// TIA Portal V17 export
// export: Created 2023-02-13T11:16:20.9592979Z, ExportSetting WithDefaults, DisplayName Totally Integrated Automation Portal, DisplayVersion V17, DisplayName TIA Portal Openness, DisplayVersion V17, DisplayName TIA Portal Teamcenter Gateway, DisplayVersion V17, DisplayName TIA Portal Version Control Interface, DisplayVersion V17, DisplayName SINAMICS Startdrive Advanced, DisplayVersion V17, DisplayName SINAMICS Startdrive G130, G150, S120, S150, SINAMICS MV, S210, DisplayVersion V17, DisplayName SINAMICS Startdrive G110M, G120, G120C, G120D, G120P, G115D, DisplayVersion V17, DisplayName STEP 7 Professional, DisplayVersion V17, DisplayName STEP 7 Safety, DisplayVersion V17, DisplayName WinCC Professional, DisplayVersion V17
DATA_BLOCK "IO Digital Blending_DB"   // DB7
VERSION : 0.1
// stored: AutoNumber true, DBAccessibleFromOPCUA true, DBAccessibleFromWebserver true, InstanceOfName IO Digital Blending, InstanceOfType FB
"IO Digital Blending"
   // VAR_INPUT
   //    Init : Bool;
   //    Reset : Bool;
   // END_VAR
   // VAR
   //    "DRP-P22.01" { S7_SetPoint := 'True'} : "Digital";
   //    "DRP-P32.01" { S7_SetPoint := 'True'} : "Digital";
   // END_VAR
BEGIN
END_DATA_BLOCK
